INTERFACE I_MoverApplication

METHOD Cycle
END_METHOD

PROPERTY P_MoverIndex : INT
GET
END_GET
SET
END_SET
END_PROPERTY

PROPERTY P_ProductData : Reference to ST_ProductData
GET
END_GET
SET
END_SET
END_PROPERTY

PROPERTY P_TrackId : UDINT
GET
END_GET
SET
END_SET
END_PROPERTY

PROPERTY std : I_XPlanarMoverStandard
GET
END_GET
SET
END_SET
END_PROPERTY

END_INTERFACE

(* stored: Version 1.1.0.1, ProductVersion 3.1.4024.9
   Itf I_MoverApplication: Id {2d233772-f0bf-4695-a678-fe38f4e7c1c5}
   Method Cycle: Id {f43fd93a-e2cb-47c2-a3de-21bdc47238e4}
   Property P_MoverIndex: Id {4f8c3075-92e1-4b10-bfa6-f4a114e4b7a1}
   Get Get: Id {3b99cd83-19d1-4af4-ab9f-5eff4d1efcb8}
   Set Set: Id {abd560e0-fa77-46be-91e3-66acff6c720a}
   Property P_ProductData: Id {3b03a1c6-796a-4d01-b444-d57076cdc9eb}
   Get Get: Id {16df046f-9c26-449c-8309-dd706c232b69}
   Set Set: Id {67002266-736a-447e-88cf-2b0fd2186e1e}
   Property P_TrackId: Id {1e1e122f-b4ed-43b3-a453-0a593fc24b6d}
   Get Get: Id {01e8f662-4981-4055-8180-6caf5d9fb045}
   Set Set: Id {cc6df96b-abb1-481a-884a-ad88396cdcc5}
   Property std: Id {05327cc5-17a4-457d-b31f-c5ae95d8b6e6}
   Get Get: Id {45bcb9f9-0a7a-4b76-8bdf-8c82272a7da1}
   Set Set: Id {e2f1fc17-80b0-4048-8c41-007948767f1a} *)
